(* PLC project  *)

PROGRAM P
  VAR  (* added by the conversion: wires and edge detectors of the diagram *)
    _ADD3_ENO : BOOL;
    _ADD3_OUT : ANY;
  END_VAR

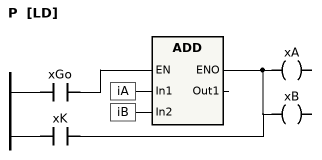
(* LD diagram, written out as Structured Text *)
_ADD3_OUT := ADD(EN := xGo, IN1 := iA, IN2 := iB, ENO => _ADD3_ENO);
xA := _ADD3_ENO;
xB := _ADD3_ENO OR xK;
END_PROGRAM
